// TIA Portal V19 export
TYPE "LEXCHANGETRAY_typeCellsMonitor"
// stored: Access Published
   STRUCT
      cellsResult : Array[0..99] of Bool;
      cellsCode : Array[0..99] of Int;
      cellSize : Int;
      nextScratchCellIndex : Int;   // 下一个要抓取电芯的索引号
   END_STRUCT;
END_TYPE
